INTERFACE ITF_TopElement1_HMI_Connector EXTENDS ITF_BaseTopElement_HMI_Connector

END_INTERFACE

(* stored: Version 1.1.0.1, ProductVersion 3.1.4024.15
   Itf ITF_TopElement1_HMI_Connector: Id {b987259f-ba74-0e29-3399-cb196a739695} *)
